RoboDK station: MESA_1.rdk

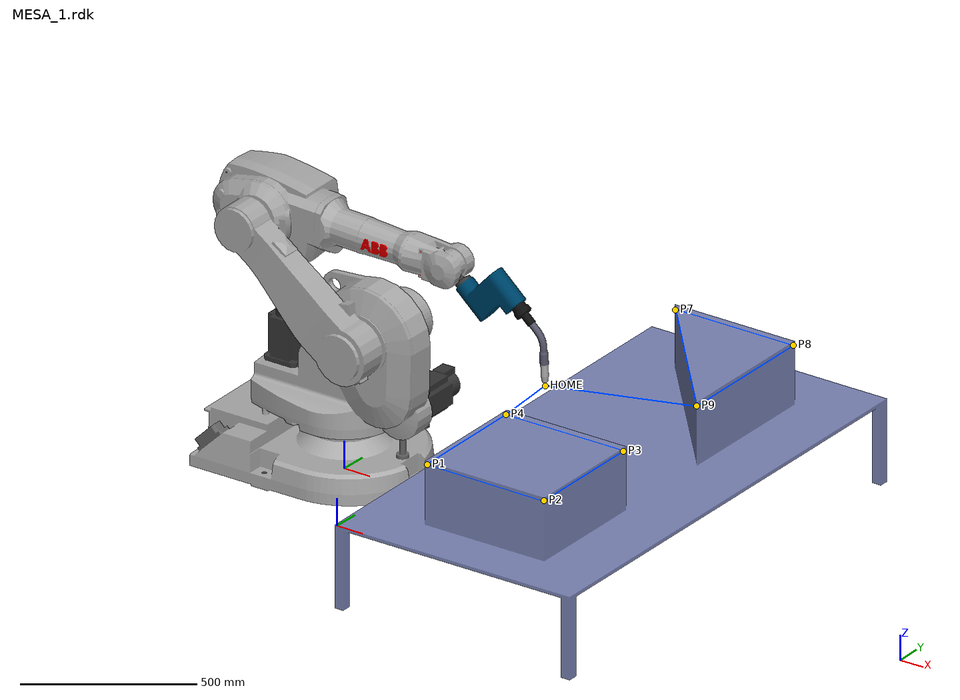
[picture v0: the station drawn from its stored meshes, robots at their saved joint values, targets as dots, program paths as lines]
Station MESA_1 (saved by RoboDK 5.9.0). Poses are relative to the parent item; angles as X-Y-Z fixed-axis rotations.
  - object mesa_1 at (1300, -750, 0) mm, rotated rx 90 ry 0 rz 90 deg, size 1560 x 460 x 810 mm, geometry from mesa_1.IGS
  - frame ABB IRB 1600-6/1.2 Base at (0, 0, 0) mm
    - robot ABB IRB 1600-6/1.2: 6 axes, payload 6 kg, reach 1200 mm, repeatability 0.05 mm, weight 250 kg
        modified DH rows (alpha deg, a mm, theta deg, d mm): 0, 0, 0, 486.5; -90, 150, -90, 0; 0, 475, 0, 0; -90, 0, 0, 600; 90, 0, 0, 0; -90, 0, 180, 65
        joint limits [-180, -90, -245, -200, -115, -400] to [180, 120, 65, 200, 115, 400]; home [0, 0, 0, 0, 0, 0]; saved at [-0.156, -54.118, 56.212, 0.18, 40.127, -0.242]
      - tool Weld gun, TCP at (-4, 0, 371.3) mm, rotated rx 0 ry 45 rz 0 deg, size 299.9 x 60 x 318.3 mm
  - frame Frame 2 at (500, -750, 260) mm
    - target HOME (Cartesian target) at (190.5, 750, 192.8) mm, rotated rx -180 ry 2.78 rz -180 deg; joints [0, -54.127, 56.211, 0, 40.136, 0] of ABB IRB 1600-6/1.2
    - target P4 (Cartesian target) at (198.19, 545.13, 185.44) mm, rotated rx -180 ry 2.78 rz 180 deg; joints [-28.817, -41.631, 51.793, 33.129, 40.778, -46.587] of ABB IRB 1600-6/1.2
    - target P1 (Cartesian target) at (201.56, 154.11, 186.7) mm, rotated rx -180 ry 2.78 rz 180 deg; joints [-57.765, -0.231, 22.212, 52.811, 51.843, -85.975] of ABB IRB 1600-6/1.2
    - target P2 (Cartesian target) at (603.16, 154.11, 185.56) mm, rotated rx -180 ry 2.78 rz 180 deg; joints [-37.472, 31.724, -16.779, 42.154, 42.169, -61.114] of ABB IRB 1600-6/1.2
    - target P3 (Cartesian target) at (603.16, 545.13, 185.56) mm, rotated rx -180 ry 2.78 rz 180 deg; joints [-14.764, 11.443, 9.685, 27.107, 24.468, -35.024] of ABB IRB 1600-6/1.2
    - target P4 (Cartesian target) at (198.19, 545.13, 185.44) mm, rotated rx -180 ry 2.78 rz 180 deg; joints [-28.817, -41.631, 51.793, 33.129, 40.778, -46.587] of ABB IRB 1600-6/1.2
    - target HOME (Cartesian target) at (190.5, 750, 192.8) mm, rotated rx -180 ry 2.78 rz -180 deg; joints [0, -54.127, 56.211, 0, 40.136, 0] of ABB IRB 1600-6/1.2
    - target P9 (Cartesian target) at (606.05, 900.61, 185.56) mm, rotated rx -180 ry 2.78 rz 180 deg; joints [10.926, 10.386, 10.912, -21.195, 22.845, 27.055] of ABB IRB 1600-6/1.2
    - target P8 (Cartesian target) at (606.05, 1376.71, 185.56) mm, rotated rx -180 ry 2.78 rz 180 deg; joints [38.772, 34.353, -20.578, -41.993, 43.881, 61.335] of ABB IRB 1600-6/1.2
    - target P7 (Cartesian target) at (202.13, 1373.97, 185.13) mm, rotated rx -180 ry 2.78 rz 180 deg; joints [58.905, 2.739, 19.347, -52.943, 52.622, 86.888] of ABB IRB 1600-6/1.2
    - target P9 (Cartesian target) at (606.05, 900.61, 185.56) mm, rotated rx -180 ry 2.78 rz 180 deg; joints [10.926, 10.386, 10.912, -21.195, 22.845, 27.055] of ABB IRB 1600-6/1.2
    - target HOME (Cartesian target) at (190.5, 750, 192.8) mm, rotated rx -180 ry 2.78 rz -180 deg; joints [0, -54.127, 56.211, 0, 40.136, 0] of ABB IRB 1600-6/1.2
  - program Prog1 (14 instructions, listed below)
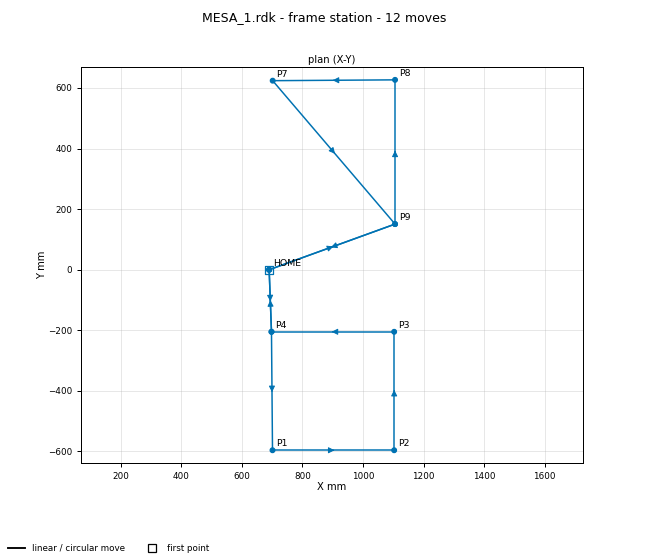
[picture p0: tool path of MESA_1.rdk in frame station, 12 of 12 moves have a stored position in this frame; points joined in program order, loops and branches not executed]

--- program Prog1 (robot ABB IRB 1600-6/1.2) ---
  Est. Ref.: Frame 2
  Est. herr: Weld gun
  MoveJ (HOME)
  MoveL (P4)
  MoveL (P1)
  MoveL (P2)
  MoveL (P3)
  MoveL (P4)
  MoveL (HOME)
  MoveL (P9)
  MoveL (P8)
  MoveL (P7)
  MoveL (P9)
  MoveL (HOME)
